TYPE "LBP_typeTMTurret"
TITLE = Tool management / Gestión de herramientas / Werkzeugverwaltung
// User data type for block LBP_TMTurret [DB73] / Tipo de dato de usuario para bloque LBP_TMTurret [DB73] / Anwender-Datentyp für Baustein LBP_TMTurret [DB73]
// stored: IsFailsafeCompliant false
   STRUCT
      IFNo : Array[1..16] of Bool;   // Schnittstelle [Nummer] aktiv / Interface [number] active / Interfaz [número] activa
      Quit : Array[1..16] of Bool;   // Quit-End durchführen / Perform Quit-End / Ejecutar Finalizar confirmación
      TIF : Array[1..16] of Struct
         Comp : Bool;   // Obligatorische Änderung / Compulsory change / Cambio obligatorio
         Perform : Bool;   // Änderung/Wechsel durchführen / Perform change / Ejecutar cambio
         f0_2 : Bool;   // Reserviert / Reserved / Reservado
         T0 : Bool;   // T0 programmiert / T0 programmed / T0 programado
         f0_4 : Bool;   // Reserviert / Reserved / Reservado
         f0_5 : Bool;   // Reserviert / Reserved / Reservado
         ManTOut : Bool;   // Handwerkzeug manuell aus Spindel entladen / Unload hand tool from spindle manually / Descargar a mano herramienta manual del cabezal
         f0_7 : Bool;   // Reserviert / Reserved / Reservado
         PerfStatusError : Bool;   // Negative Quittung / Negative acknowledge / Confirmación negativa
         n1_1 : Bool;   // Reserviert / Reserved / Reservado
         n1_2 : Bool;   // Reserviert / Reserved / Reservado
         n1_3 : Bool;   // Reserviert / Reserved / Reservado
         n1_4 : Bool;   // Reserviert / Reserved / Reservado
         n1_5 : Bool;   // Reserviert / Reserved / Reservado
         n1_6 : Bool;   // Reserviert / Reserved / Reservado
         DataInDB1073 : Bool;   // Multitool-Daten gespeichert in DB1073 / Multitool data stored in DB1073 / Datos Multitool guardados en DB1073
         Channel : Byte;   // Zugeordneter Kanal / Assigned channel / Canal asignado
         TMNo : Byte;   // Werkzeug-Verwaltungsnummer / Tool management number / Número de gestión de herramientas
         VdiTcp0 : DInt;   // Freie Anwendervariable 0 / User parameter 0 / Parámetro de usuario 0
         VdiTcp1 : DInt;   // Freie Anwendervariable 1 / User parameter 1 / Parámetro de usuario 1
         VdiTcp2 : DInt;   // Freie Anwendervariable 2 / User parameter 2 / Parámetro de usuario 2
         BufferIdent : Int;   // Reserviert (Puffer-Identifikation) / Reserved (buffer identification) / Reservado (identificación de búfer)
         BufferNo : Int;   // Rel. Platz im Puffer (res.) / Rel. location in buffer (res.) / Puesto rel. en búfer (res.)
         SMag : Int;   // Magazin-Nummer des Revolvers / Magazine number of turret / Número de almacén del revólver
         SLoc : Int;   // Platznummer für neues Werkzeug / Location number for new tool / Número de puesto para nueva herramienta
         TMag : Int;   // Magazin-Nummer des Revolvers (res.) / Magazine number of turret (res.) / Número de almacén del revólver (res.)
         TLoc : Int;   // Platznummer für vorheriges Werkzeug / Location number for previous tool / Número de puesto para herramienta previa
         LocType : Int;   // Werkzeug neu: Platzart / Tool new: location type / Herramienta nueva: tipo de puesto
         SLeft : Int;   // Werkeug neu: Größe links / Tool new: size left / Herramienta nueva: tamaño izquierda
         SRight : Int;   // Werkeug neu: Größe rechts / Tool new: size right / Herramienta nueva: tamaño derecha
         STop : Int;   // Werkeug neu: Größe oben / Tool new: size top / Herramienta nueva: tamaño arriba
         SBottom : Int;   // Werkeug neu: Größe unten / Tool new: size bottom / Herramienta nueva: tamaño abajo
         TInBuffer : Bool;   // ID für Werkzeuge im Puffer / ID for tools in buffer / ID para herramientas en búfer
         IgnoreDisabled : Bool;   // Deaktiviert ignorieren / Ignore disabled / Ignorar desactivado
         Unload : Bool;   // Zu entladen / To be unloaded / Por descargar
         Load : Bool;   // Zu laden / To be loaded / Por cargar
         MasterTool : Bool;   // Master-Werkzeug / Master tool / Herramienta maestra
         n38_5 : Bool;   // Reserviert / Reserved / Reservado
         Exchange_1to1 : Bool;   // 1:1 Austausch / 1:1 exchange / Cambio 1:1
         HandTool : Bool;   // Handwerkzeug / Hand tool / Herramienta manual
         Active : Bool;   // Aktives Werkzeug / Active tool / Herramienta activa
         Enabled : Bool;   // Werkzeug aktiviert / Tool enabled / Herramienta activada
         Disabled : Bool;   // Werkzeug deaktiviert / Tool disabled / Herramienta desactivada
         Measured : Bool;   // Werkzeug gemessen / Tool measured / Herramienta medida
         Prewarn : Bool;   // Vorwarnungsgrenze erreicht / Prewarning limit reached / Límite de prealarma alcanzado
         Change : Bool;   // Werkzeug wird gewechselt / Tool being changed / Sustituyendo herramienta
         FixedLoc : Bool;   // Werkzeug-Festplatz codiert / Tool fixed location coded / Puesto fijo de herramienta codificado
         Used : Bool;   // Werkzeug war in Gebrauch / Tool was in use / La herramienta estaba en uso
         TNo : Int;   // Werkzeug neu: WZ-Nummer / Tool new: T number / Herramienta nueva: n.º herramienta
         MyPlace : Int;   // Originalplatz des neuen Werkzeugs / Original location of new tool / Puesto de origen de la nueva herramienta
      END_STRUCT;
   END_STRUCT;
   // // TIF[2].Comp : Obligatorische Änderung / Compulsory change / Cambio obligatorio
   // // TIF[3].Comp : Obligatorische Änderung / Compulsory change / Cambio obligatorio
   // // TIF[4].Comp : Obligatorische Änderung / Compulsory change / Cambio obligatorio
   // // TIF[5].Comp : Obligatorische Änderung / Compulsory change / Cambio obligatorio
   // // TIF[6].Comp : Obligatorische Änderung / Compulsory change / Cambio obligatorio
   // // TIF[7].Comp : Obligatorische Änderung / Compulsory change / Cambio obligatorio
   // // TIF[8].Comp : Obligatorische Änderung / Compulsory change / Cambio obligatorio
   // // TIF[9].Comp : Obligatorische Änderung / Compulsory change / Cambio obligatorio
   // // TIF[10].Comp : Obligatorische Änderung / Compulsory change / Cambio obligatorio
   // // TIF[11].Comp : Obligatorische Änderung / Compulsory change / Cambio obligatorio
   // // TIF[12].Comp : Obligatorische Änderung / Compulsory change / Cambio obligatorio
   // // TIF[13].Comp : Obligatorische Änderung / Compulsory change / Cambio obligatorio
   // // TIF[14].Comp : Obligatorische Änderung / Compulsory change / Cambio obligatorio
   // // TIF[15].Comp : Obligatorische Änderung / Compulsory change / Cambio obligatorio
   // // TIF[16].Comp : Obligatorische Änderung / Compulsory change / Cambio obligatorio
   // // TIF[2].Perform : Änderung/Wechsel durchführen / Perform change / Ejecutar cambio
   // // TIF[3].Perform : Änderung/Wechsel durchführen / Perform change / Ejecutar cambio
   // // TIF[4].Perform : Änderung/Wechsel durchführen / Perform change / Ejecutar cambio
   // // TIF[5].Perform : Änderung/Wechsel durchführen / Perform change / Ejecutar cambio
   // // TIF[6].Perform : Änderung/Wechsel durchführen / Perform change / Ejecutar cambio
   // // TIF[7].Perform : Änderung/Wechsel durchführen / Perform change / Ejecutar cambio
   // // TIF[8].Perform : Änderung/Wechsel durchführen / Perform change / Ejecutar cambio
   // // TIF[9].Perform : Änderung/Wechsel durchführen / Perform change / Ejecutar cambio
   // // TIF[10].Perform : Änderung/Wechsel durchführen / Perform change / Ejecutar cambio
   // // TIF[11].Perform : Änderung/Wechsel durchführen / Perform change / Ejecutar cambio
   // // TIF[12].Perform : Änderung/Wechsel durchführen / Perform change / Ejecutar cambio
   // // TIF[13].Perform : Änderung/Wechsel durchführen / Perform change / Ejecutar cambio
   // // TIF[14].Perform : Änderung/Wechsel durchführen / Perform change / Ejecutar cambio
   // // TIF[15].Perform : Änderung/Wechsel durchführen / Perform change / Ejecutar cambio
   // // TIF[16].Perform : Änderung/Wechsel durchführen / Perform change / Ejecutar cambio
   // // TIF[2].f0_2 : Reserviert / Reserved / Reservado
   // // TIF[3].f0_2 : Reserviert / Reserved / Reservado
   // // TIF[4].f0_2 : Reserviert / Reserved / Reservado
   // // TIF[5].f0_2 : Reserviert / Reserved / Reservado
   // // TIF[6].f0_2 : Reserviert / Reserved / Reservado
   // // TIF[7].f0_2 : Reserviert / Reserved / Reservado
   // // TIF[8].f0_2 : Reserviert / Reserved / Reservado
   // // TIF[9].f0_2 : Reserviert / Reserved / Reservado
   // // TIF[10].f0_2 : Reserviert / Reserved / Reservado
   // // TIF[11].f0_2 : Reserviert / Reserved / Reservado
   // // TIF[12].f0_2 : Reserviert / Reserved / Reservado
   // // TIF[13].f0_2 : Reserviert / Reserved / Reservado
   // // TIF[14].f0_2 : Reserviert / Reserved / Reservado
   // // TIF[15].f0_2 : Reserviert / Reserved / Reservado
   // // TIF[16].f0_2 : Reserviert / Reserved / Reservado
   // // TIF[2].T0 : T0 programmiert / T0 programmed / T0 programado
   // // TIF[3].T0 : T0 programmiert / T0 programmed / T0 programado
   // // TIF[4].T0 : T0 programmiert / T0 programmed / T0 programado
   // // TIF[5].T0 : T0 programmiert / T0 programmed / T0 programado
   // // TIF[6].T0 : T0 programmiert / T0 programmed / T0 programado
   // // TIF[7].T0 : T0 programmiert / T0 programmed / T0 programado
   // // TIF[8].T0 : T0 programmiert / T0 programmed / T0 programado
   // // TIF[9].T0 : T0 programmiert / T0 programmed / T0 programado
   // // TIF[10].T0 : T0 programmiert / T0 programmed / T0 programado
   // // TIF[11].T0 : T0 programmiert / T0 programmed / T0 programado
   // // TIF[12].T0 : T0 programmiert / T0 programmed / T0 programado
   // // TIF[13].T0 : T0 programmiert / T0 programmed / T0 programado
   // // TIF[14].T0 : T0 programmiert / T0 programmed / T0 programado
   // // TIF[15].T0 : T0 programmiert / T0 programmed / T0 programado
   // // TIF[16].T0 : T0 programmiert / T0 programmed / T0 programado
   // // TIF[2].f0_4 : Reserviert / Reserved / Reservado
   // // TIF[3].f0_4 : Reserviert / Reserved / Reservado
   // // TIF[4].f0_4 : Reserviert / Reserved / Reservado
   // // TIF[5].f0_4 : Reserviert / Reserved / Reservado
   // // TIF[6].f0_4 : Reserviert / Reserved / Reservado
   // // TIF[7].f0_4 : Reserviert / Reserved / Reservado
   // // TIF[8].f0_4 : Reserviert / Reserved / Reservado
   // // TIF[9].f0_4 : Reserviert / Reserved / Reservado
   // // TIF[10].f0_4 : Reserviert / Reserved / Reservado
   // // TIF[11].f0_4 : Reserviert / Reserved / Reservado
   // // TIF[12].f0_4 : Reserviert / Reserved / Reservado
   // // TIF[13].f0_4 : Reserviert / Reserved / Reservado
   // // TIF[14].f0_4 : Reserviert / Reserved / Reservado
   // // TIF[15].f0_4 : Reserviert / Reserved / Reservado
   // // TIF[16].f0_4 : Reserviert / Reserved / Reservado
   // // TIF[2].f0_5 : Reserviert / Reserved / Reservado
   // // TIF[3].f0_5 : Reserviert / Reserved / Reservado
   // // TIF[4].f0_5 : Reserviert / Reserved / Reservado
   // // TIF[5].f0_5 : Reserviert / Reserved / Reservado
   // // TIF[6].f0_5 : Reserviert / Reserved / Reservado
   // // TIF[7].f0_5 : Reserviert / Reserved / Reservado
   // // TIF[8].f0_5 : Reserviert / Reserved / Reservado
   // // TIF[9].f0_5 : Reserviert / Reserved / Reservado
   // // TIF[10].f0_5 : Reserviert / Reserved / Reservado
   // // TIF[11].f0_5 : Reserviert / Reserved / Reservado
   // // TIF[12].f0_5 : Reserviert / Reserved / Reservado
   // // TIF[13].f0_5 : Reserviert / Reserved / Reservado
   // // TIF[14].f0_5 : Reserviert / Reserved / Reservado
   // // TIF[15].f0_5 : Reserviert / Reserved / Reservado
   // // TIF[16].f0_5 : Reserviert / Reserved / Reservado
   // // TIF[2].ManTOut : Handwerkzeug manuell aus Spindel entladen / Unload hand tool from spindle manually / Descargar a mano herramienta manual del cabezal
   // // TIF[3].ManTOut : Handwerkzeug manuell aus Spindel entladen / Unload hand tool from spindle manually / Descargar a mano herramienta manual del cabezal
   // // TIF[4].ManTOut : Handwerkzeug manuell aus Spindel entladen / Unload hand tool from spindle manually / Descargar a mano herramienta manual del cabezal
   // // TIF[5].ManTOut : Handwerkzeug manuell aus Spindel entladen / Unload hand tool from spindle manually / Descargar a mano herramienta manual del cabezal
   // // TIF[6].ManTOut : Handwerkzeug manuell aus Spindel entladen / Unload hand tool from spindle manually / Descargar a mano herramienta manual del cabezal
   // // TIF[7].ManTOut : Handwerkzeug manuell aus Spindel entladen / Unload hand tool from spindle manually / Descargar a mano herramienta manual del cabezal
   // // TIF[8].ManTOut : Handwerkzeug manuell aus Spindel entladen / Unload hand tool from spindle manually / Descargar a mano herramienta manual del cabezal
   // // TIF[9].ManTOut : Handwerkzeug manuell aus Spindel entladen / Unload hand tool from spindle manually / Descargar a mano herramienta manual del cabezal
   // // TIF[10].ManTOut : Handwerkzeug manuell aus Spindel entladen / Unload hand tool from spindle manually / Descargar a mano herramienta manual del cabezal
   // // TIF[11].ManTOut : Handwerkzeug manuell aus Spindel entladen / Unload hand tool from spindle manually / Descargar a mano herramienta manual del cabezal
   // // TIF[12].ManTOut : Handwerkzeug manuell aus Spindel entladen / Unload hand tool from spindle manually / Descargar a mano herramienta manual del cabezal
   // // TIF[13].ManTOut : Handwerkzeug manuell aus Spindel entladen / Unload hand tool from spindle manually / Descargar a mano herramienta manual del cabezal
   // // TIF[14].ManTOut : Handwerkzeug manuell aus Spindel entladen / Unload hand tool from spindle manually / Descargar a mano herramienta manual del cabezal
   // // TIF[15].ManTOut : Handwerkzeug manuell aus Spindel entladen / Unload hand tool from spindle manually / Descargar a mano herramienta manual del cabezal
   // // TIF[16].ManTOut : Handwerkzeug manuell aus Spindel entladen / Unload hand tool from spindle manually / Descargar a mano herramienta manual del cabezal
   // // TIF[2].f0_7 : Reserviert / Reserved / Reservado
   // // TIF[3].f0_7 : Reserviert / Reserved / Reservado
   // // TIF[4].f0_7 : Reserviert / Reserved / Reservado
   // // TIF[5].f0_7 : Reserviert / Reserved / Reservado
   // // TIF[6].f0_7 : Reserviert / Reserved / Reservado
   // // TIF[7].f0_7 : Reserviert / Reserved / Reservado
   // // TIF[8].f0_7 : Reserviert / Reserved / Reservado
   // // TIF[9].f0_7 : Reserviert / Reserved / Reservado
   // // TIF[10].f0_7 : Reserviert / Reserved / Reservado
   // // TIF[11].f0_7 : Reserviert / Reserved / Reservado
   // // TIF[12].f0_7 : Reserviert / Reserved / Reservado
   // // TIF[13].f0_7 : Reserviert / Reserved / Reservado
   // // TIF[14].f0_7 : Reserviert / Reserved / Reservado
   // // TIF[15].f0_7 : Reserviert / Reserved / Reservado
   // // TIF[16].f0_7 : Reserviert / Reserved / Reservado
   // // TIF[2].PerfStatusError : Negative Quittung / Negative acknowledge / Confirmación negativa
   // // TIF[3].PerfStatusError : Negative Quittung / Negative acknowledge / Confirmación negativa
   // // TIF[4].PerfStatusError : Negative Quittung / Negative acknowledge / Confirmación negativa
   // // TIF[5].PerfStatusError : Negative Quittung / Negative acknowledge / Confirmación negativa
   // // TIF[6].PerfStatusError : Negative Quittung / Negative acknowledge / Confirmación negativa
   // // TIF[7].PerfStatusError : Negative Quittung / Negative acknowledge / Confirmación negativa
   // // TIF[8].PerfStatusError : Negative Quittung / Negative acknowledge / Confirmación negativa
   // // TIF[9].PerfStatusError : Negative Quittung / Negative acknowledge / Confirmación negativa
   // // TIF[10].PerfStatusError : Negative Quittung / Negative acknowledge / Confirmación negativa
   // // TIF[11].PerfStatusError : Negative Quittung / Negative acknowledge / Confirmación negativa
   // // TIF[12].PerfStatusError : Negative Quittung / Negative acknowledge / Confirmación negativa
   // // TIF[13].PerfStatusError : Negative Quittung / Negative acknowledge / Confirmación negativa
   // // TIF[14].PerfStatusError : Negative Quittung / Negative acknowledge / Confirmación negativa
   // // TIF[15].PerfStatusError : Negative Quittung / Negative acknowledge / Confirmación negativa
   // // TIF[16].PerfStatusError : Negative Quittung / Negative acknowledge / Confirmación negativa
   // // TIF[2].n1_1 : Reserviert / Reserved / Reservado
   // // TIF[3].n1_1 : Reserviert / Reserved / Reservado
   // // TIF[4].n1_1 : Reserviert / Reserved / Reservado
   // // TIF[5].n1_1 : Reserviert / Reserved / Reservado
   // // TIF[6].n1_1 : Reserviert / Reserved / Reservado
   // // TIF[7].n1_1 : Reserviert / Reserved / Reservado
   // // TIF[8].n1_1 : Reserviert / Reserved / Reservado
   // // TIF[9].n1_1 : Reserviert / Reserved / Reservado
   // // TIF[10].n1_1 : Reserviert / Reserved / Reservado
   // // TIF[11].n1_1 : Reserviert / Reserved / Reservado
   // // TIF[12].n1_1 : Reserviert / Reserved / Reservado
   // // TIF[13].n1_1 : Reserviert / Reserved / Reservado
   // // TIF[14].n1_1 : Reserviert / Reserved / Reservado
   // // TIF[15].n1_1 : Reserviert / Reserved / Reservado
   // // TIF[16].n1_1 : Reserviert / Reserved / Reservado
   // // TIF[2].n1_2 : Reserviert / Reserved / Reservado
   // // TIF[3].n1_2 : Reserviert / Reserved / Reservado
   // // TIF[4].n1_2 : Reserviert / Reserved / Reservado
   // // TIF[5].n1_2 : Reserviert / Reserved / Reservado
   // // TIF[6].n1_2 : Reserviert / Reserved / Reservado
   // // TIF[7].n1_2 : Reserviert / Reserved / Reservado
   // // TIF[8].n1_2 : Reserviert / Reserved / Reservado
   // // TIF[9].n1_2 : Reserviert / Reserved / Reservado
   // // TIF[10].n1_2 : Reserviert / Reserved / Reservado
   // // TIF[11].n1_2 : Reserviert / Reserved / Reservado
   // // TIF[12].n1_2 : Reserviert / Reserved / Reservado
   // // TIF[13].n1_2 : Reserviert / Reserved / Reservado
   // // TIF[14].n1_2 : Reserviert / Reserved / Reservado
   // // TIF[15].n1_2 : Reserviert / Reserved / Reservado
   // // TIF[16].n1_2 : Reserviert / Reserved / Reservado
   // // TIF[2].n1_3 : Reserviert / Reserved / Reservado
   // // TIF[3].n1_3 : Reserviert / Reserved / Reservado
   // // TIF[4].n1_3 : Reserviert / Reserved / Reservado
   // // TIF[5].n1_3 : Reserviert / Reserved / Reservado
   // // TIF[6].n1_3 : Reserviert / Reserved / Reservado
   // // TIF[7].n1_3 : Reserviert / Reserved / Reservado
   // // TIF[8].n1_3 : Reserviert / Reserved / Reservado
   // // TIF[9].n1_3 : Reserviert / Reserved / Reservado
   // // TIF[10].n1_3 : Reserviert / Reserved / Reservado
   // // TIF[11].n1_3 : Reserviert / Reserved / Reservado
   // // TIF[12].n1_3 : Reserviert / Reserved / Reservado
   // // TIF[13].n1_3 : Reserviert / Reserved / Reservado
   // // TIF[14].n1_3 : Reserviert / Reserved / Reservado
   // // TIF[15].n1_3 : Reserviert / Reserved / Reservado
   // // TIF[16].n1_3 : Reserviert / Reserved / Reservado
   // // TIF[2].n1_4 : Reserviert / Reserved / Reservado
   // // TIF[3].n1_4 : Reserviert / Reserved / Reservado
   // // TIF[4].n1_4 : Reserviert / Reserved / Reservado
   // // TIF[5].n1_4 : Reserviert / Reserved / Reservado
   // // TIF[6].n1_4 : Reserviert / Reserved / Reservado
   // // TIF[7].n1_4 : Reserviert / Reserved / Reservado
   // // TIF[8].n1_4 : Reserviert / Reserved / Reservado
   // // TIF[9].n1_4 : Reserviert / Reserved / Reservado
   // // TIF[10].n1_4 : Reserviert / Reserved / Reservado
   // // TIF[11].n1_4 : Reserviert / Reserved / Reservado
   // // TIF[12].n1_4 : Reserviert / Reserved / Reservado
   // // TIF[13].n1_4 : Reserviert / Reserved / Reservado
   // // TIF[14].n1_4 : Reserviert / Reserved / Reservado
   // // TIF[15].n1_4 : Reserviert / Reserved / Reservado
   // // TIF[16].n1_4 : Reserviert / Reserved / Reservado
   // // TIF[2].n1_5 : Reserviert / Reserved / Reservado
   // // TIF[3].n1_5 : Reserviert / Reserved / Reservado
   // // TIF[4].n1_5 : Reserviert / Reserved / Reservado
   // // TIF[5].n1_5 : Reserviert / Reserved / Reservado
   // // TIF[6].n1_5 : Reserviert / Reserved / Reservado
   // // TIF[7].n1_5 : Reserviert / Reserved / Reservado
   // // TIF[8].n1_5 : Reserviert / Reserved / Reservado
   // // TIF[9].n1_5 : Reserviert / Reserved / Reservado
   // // TIF[10].n1_5 : Reserviert / Reserved / Reservado
   // // TIF[11].n1_5 : Reserviert / Reserved / Reservado
   // // TIF[12].n1_5 : Reserviert / Reserved / Reservado
   // // TIF[13].n1_5 : Reserviert / Reserved / Reservado
   // // TIF[14].n1_5 : Reserviert / Reserved / Reservado
   // // TIF[15].n1_5 : Reserviert / Reserved / Reservado
   // // TIF[16].n1_5 : Reserviert / Reserved / Reservado
   // // TIF[2].n1_6 : Reserviert / Reserved / Reservado
   // // TIF[3].n1_6 : Reserviert / Reserved / Reservado
   // // TIF[4].n1_6 : Reserviert / Reserved / Reservado
   // // TIF[5].n1_6 : Reserviert / Reserved / Reservado
   // // TIF[6].n1_6 : Reserviert / Reserved / Reservado
   // // TIF[7].n1_6 : Reserviert / Reserved / Reservado
   // // TIF[8].n1_6 : Reserviert / Reserved / Reservado
   // // TIF[9].n1_6 : Reserviert / Reserved / Reservado
   // // TIF[10].n1_6 : Reserviert / Reserved / Reservado
   // // TIF[11].n1_6 : Reserviert / Reserved / Reservado
   // // TIF[12].n1_6 : Reserviert / Reserved / Reservado
   // // TIF[13].n1_6 : Reserviert / Reserved / Reservado
   // // TIF[14].n1_6 : Reserviert / Reserved / Reservado
   // // TIF[15].n1_6 : Reserviert / Reserved / Reservado
   // // TIF[16].n1_6 : Reserviert / Reserved / Reservado
   // // TIF[2].DataInDB1073 : Multitool-Daten gespeichert in DB1073 / Multitool data stored in DB1073 / Datos Multitool guardados en DB1073
   // // TIF[3].DataInDB1073 : Multitool-Daten gespeichert in DB1073 / Multitool data stored in DB1073 / Datos Multitool guardados en DB1073
   // // TIF[4].DataInDB1073 : Multitool-Daten gespeichert in DB1073 / Multitool data stored in DB1073 / Datos Multitool guardados en DB1073
   // // TIF[5].DataInDB1073 : Multitool-Daten gespeichert in DB1073 / Multitool data stored in DB1073 / Datos Multitool guardados en DB1073
   // // TIF[6].DataInDB1073 : Multitool-Daten gespeichert in DB1073 / Multitool data stored in DB1073 / Datos Multitool guardados en DB1073
   // // TIF[7].DataInDB1073 : Multitool-Daten gespeichert in DB1073 / Multitool data stored in DB1073 / Datos Multitool guardados en DB1073
   // // TIF[8].DataInDB1073 : Multitool-Daten gespeichert in DB1073 / Multitool data stored in DB1073 / Datos Multitool guardados en DB1073
   // // TIF[9].DataInDB1073 : Multitool-Daten gespeichert in DB1073 / Multitool data stored in DB1073 / Datos Multitool guardados en DB1073
   // // TIF[10].DataInDB1073 : Multitool-Daten gespeichert in DB1073 / Multitool data stored in DB1073 / Datos Multitool guardados en DB1073
   // // TIF[11].DataInDB1073 : Multitool-Daten gespeichert in DB1073 / Multitool data stored in DB1073 / Datos Multitool guardados en DB1073
   // // TIF[12].DataInDB1073 : Multitool-Daten gespeichert in DB1073 / Multitool data stored in DB1073 / Datos Multitool guardados en DB1073
   // // TIF[13].DataInDB1073 : Multitool-Daten gespeichert in DB1073 / Multitool data stored in DB1073 / Datos Multitool guardados en DB1073
   // // TIF[14].DataInDB1073 : Multitool-Daten gespeichert in DB1073 / Multitool data stored in DB1073 / Datos Multitool guardados en DB1073
   // // TIF[15].DataInDB1073 : Multitool-Daten gespeichert in DB1073 / Multitool data stored in DB1073 / Datos Multitool guardados en DB1073
   // // TIF[16].DataInDB1073 : Multitool-Daten gespeichert in DB1073 / Multitool data stored in DB1073 / Datos Multitool guardados en DB1073
   // // TIF[2].Channel : Zugeordneter Kanal / Assigned channel / Canal asignado
   // // TIF[3].Channel : Zugeordneter Kanal / Assigned channel / Canal asignado
   // // TIF[4].Channel : Zugeordneter Kanal / Assigned channel / Canal asignado
   // // TIF[5].Channel : Zugeordneter Kanal / Assigned channel / Canal asignado
   // // TIF[6].Channel : Zugeordneter Kanal / Assigned channel / Canal asignado
   // // TIF[7].Channel : Zugeordneter Kanal / Assigned channel / Canal asignado
   // // TIF[8].Channel : Zugeordneter Kanal / Assigned channel / Canal asignado
   // // TIF[9].Channel : Zugeordneter Kanal / Assigned channel / Canal asignado
   // // TIF[10].Channel : Zugeordneter Kanal / Assigned channel / Canal asignado
   // // TIF[11].Channel : Zugeordneter Kanal / Assigned channel / Canal asignado
   // // TIF[12].Channel : Zugeordneter Kanal / Assigned channel / Canal asignado
   // // TIF[13].Channel : Zugeordneter Kanal / Assigned channel / Canal asignado
   // // TIF[14].Channel : Zugeordneter Kanal / Assigned channel / Canal asignado
   // // TIF[15].Channel : Zugeordneter Kanal / Assigned channel / Canal asignado
   // // TIF[16].Channel : Zugeordneter Kanal / Assigned channel / Canal asignado
   // // TIF[2].TMNo : Werkzeug-Verwaltungsnummer / Tool management number / Número de gestión de herramientas
   // // TIF[3].TMNo : Werkzeug-Verwaltungsnummer / Tool management number / Número de gestión de herramientas
   // // TIF[4].TMNo : Werkzeug-Verwaltungsnummer / Tool management number / Número de gestión de herramientas
   // // TIF[5].TMNo : Werkzeug-Verwaltungsnummer / Tool management number / Número de gestión de herramientas
   // // TIF[6].TMNo : Werkzeug-Verwaltungsnummer / Tool management number / Número de gestión de herramientas
   // // TIF[7].TMNo : Werkzeug-Verwaltungsnummer / Tool management number / Número de gestión de herramientas
   // // TIF[8].TMNo : Werkzeug-Verwaltungsnummer / Tool management number / Número de gestión de herramientas
   // // TIF[9].TMNo : Werkzeug-Verwaltungsnummer / Tool management number / Número de gestión de herramientas
   // // TIF[10].TMNo : Werkzeug-Verwaltungsnummer / Tool management number / Número de gestión de herramientas
   // // TIF[11].TMNo : Werkzeug-Verwaltungsnummer / Tool management number / Número de gestión de herramientas
   // // TIF[12].TMNo : Werkzeug-Verwaltungsnummer / Tool management number / Número de gestión de herramientas
   // // TIF[13].TMNo : Werkzeug-Verwaltungsnummer / Tool management number / Número de gestión de herramientas
   // // TIF[14].TMNo : Werkzeug-Verwaltungsnummer / Tool management number / Número de gestión de herramientas
   // // TIF[15].TMNo : Werkzeug-Verwaltungsnummer / Tool management number / Número de gestión de herramientas
   // // TIF[16].TMNo : Werkzeug-Verwaltungsnummer / Tool management number / Número de gestión de herramientas
   // // TIF[2].VdiTcp0 : Freie Anwendervariable 0 / User parameter 0 / Parámetro de usuario 0
   // // TIF[3].VdiTcp0 : Freie Anwendervariable 0 / User parameter 0 / Parámetro de usuario 0
   // // TIF[4].VdiTcp0 : Freie Anwendervariable 0 / User parameter 0 / Parámetro de usuario 0
   // // TIF[5].VdiTcp0 : Freie Anwendervariable 0 / User parameter 0 / Parámetro de usuario 0
   // // TIF[6].VdiTcp0 : Freie Anwendervariable 0 / User parameter 0 / Parámetro de usuario 0
   // // TIF[7].VdiTcp0 : Freie Anwendervariable 0 / User parameter 0 / Parámetro de usuario 0
   // // TIF[8].VdiTcp0 : Freie Anwendervariable 0 / User parameter 0 / Parámetro de usuario 0
   // // TIF[9].VdiTcp0 : Freie Anwendervariable 0 / User parameter 0 / Parámetro de usuario 0
   // // TIF[10].VdiTcp0 : Freie Anwendervariable 0 / User parameter 0 / Parámetro de usuario 0
   // // TIF[11].VdiTcp0 : Freie Anwendervariable 0 / User parameter 0 / Parámetro de usuario 0
   // // TIF[12].VdiTcp0 : Freie Anwendervariable 0 / User parameter 0 / Parámetro de usuario 0
   // // TIF[13].VdiTcp0 : Freie Anwendervariable 0 / User parameter 0 / Parámetro de usuario 0
   // // TIF[14].VdiTcp0 : Freie Anwendervariable 0 / User parameter 0 / Parámetro de usuario 0
   // // TIF[15].VdiTcp0 : Freie Anwendervariable 0 / User parameter 0 / Parámetro de usuario 0
   // // TIF[16].VdiTcp0 : Freie Anwendervariable 0 / User parameter 0 / Parámetro de usuario 0
   // // TIF[2].VdiTcp1 : Freie Anwendervariable 1 / User parameter 1 / Parámetro de usuario 1
   // // TIF[3].VdiTcp1 : Freie Anwendervariable 1 / User parameter 1 / Parámetro de usuario 1
   // // TIF[4].VdiTcp1 : Freie Anwendervariable 1 / User parameter 1 / Parámetro de usuario 1
   // // TIF[5].VdiTcp1 : Freie Anwendervariable 1 / User parameter 1 / Parámetro de usuario 1
   // // TIF[6].VdiTcp1 : Freie Anwendervariable 1 / User parameter 1 / Parámetro de usuario 1
   // // TIF[7].VdiTcp1 : Freie Anwendervariable 1 / User parameter 1 / Parámetro de usuario 1
   // // TIF[8].VdiTcp1 : Freie Anwendervariable 1 / User parameter 1 / Parámetro de usuario 1
   // // TIF[9].VdiTcp1 : Freie Anwendervariable 1 / User parameter 1 / Parámetro de usuario 1
   // // TIF[10].VdiTcp1 : Freie Anwendervariable 1 / User parameter 1 / Parámetro de usuario 1
   // // TIF[11].VdiTcp1 : Freie Anwendervariable 1 / User parameter 1 / Parámetro de usuario 1
   // // TIF[12].VdiTcp1 : Freie Anwendervariable 1 / User parameter 1 / Parámetro de usuario 1
   // // TIF[13].VdiTcp1 : Freie Anwendervariable 1 / User parameter 1 / Parámetro de usuario 1
   // // TIF[14].VdiTcp1 : Freie Anwendervariable 1 / User parameter 1 / Parámetro de usuario 1
   // // TIF[15].VdiTcp1 : Freie Anwendervariable 1 / User parameter 1 / Parámetro de usuario 1
   // // TIF[16].VdiTcp1 : Freie Anwendervariable 1 / User parameter 1 / Parámetro de usuario 1
   // // TIF[2].VdiTcp2 : Freie Anwendervariable 2 / User parameter 2 / Parámetro de usuario 2
   // // TIF[3].VdiTcp2 : Freie Anwendervariable 2 / User parameter 2 / Parámetro de usuario 2
   // // TIF[4].VdiTcp2 : Freie Anwendervariable 2 / User parameter 2 / Parámetro de usuario 2
   // // TIF[5].VdiTcp2 : Freie Anwendervariable 2 / User parameter 2 / Parámetro de usuario 2
   // // TIF[6].VdiTcp2 : Freie Anwendervariable 2 / User parameter 2 / Parámetro de usuario 2
   // // TIF[7].VdiTcp2 : Freie Anwendervariable 2 / User parameter 2 / Parámetro de usuario 2
   // // TIF[8].VdiTcp2 : Freie Anwendervariable 2 / User parameter 2 / Parámetro de usuario 2
   // // TIF[9].VdiTcp2 : Freie Anwendervariable 2 / User parameter 2 / Parámetro de usuario 2
   // // TIF[10].VdiTcp2 : Freie Anwendervariable 2 / User parameter 2 / Parámetro de usuario 2
   // // TIF[11].VdiTcp2 : Freie Anwendervariable 2 / User parameter 2 / Parámetro de usuario 2
   // // TIF[12].VdiTcp2 : Freie Anwendervariable 2 / User parameter 2 / Parámetro de usuario 2
   // // TIF[13].VdiTcp2 : Freie Anwendervariable 2 / User parameter 2 / Parámetro de usuario 2
   // // TIF[14].VdiTcp2 : Freie Anwendervariable 2 / User parameter 2 / Parámetro de usuario 2
   // // TIF[15].VdiTcp2 : Freie Anwendervariable 2 / User parameter 2 / Parámetro de usuario 2
   // // TIF[16].VdiTcp2 : Freie Anwendervariable 2 / User parameter 2 / Parámetro de usuario 2
   // // TIF[2].BufferIdent : Reserviert (Puffer-Identifikation) / Reserved (buffer identification) / Reservado (identificación de búfer)
   // // TIF[3].BufferIdent : Reserviert (Puffer-Identifikation) / Reserved (buffer identification) / Reservado (identificación de búfer)
   // // TIF[4].BufferIdent : Reserviert (Puffer-Identifikation) / Reserved (buffer identification) / Reservado (identificación de búfer)
   // // TIF[5].BufferIdent : Reserviert (Puffer-Identifikation) / Reserved (buffer identification) / Reservado (identificación de búfer)
   // // TIF[6].BufferIdent : Reserviert (Puffer-Identifikation) / Reserved (buffer identification) / Reservado (identificación de búfer)
   // // TIF[7].BufferIdent : Reserviert (Puffer-Identifikation) / Reserved (buffer identification) / Reservado (identificación de búfer)
   // // TIF[8].BufferIdent : Reserviert (Puffer-Identifikation) / Reserved (buffer identification) / Reservado (identificación de búfer)
   // // TIF[9].BufferIdent : Reserviert (Puffer-Identifikation) / Reserved (buffer identification) / Reservado (identificación de búfer)
   // // TIF[10].BufferIdent : Reserviert (Puffer-Identifikation) / Reserved (buffer identification) / Reservado (identificación de búfer)
   // // TIF[11].BufferIdent : Reserviert (Puffer-Identifikation) / Reserved (buffer identification) / Reservado (identificación de búfer)
   // // TIF[12].BufferIdent : Reserviert (Puffer-Identifikation) / Reserved (buffer identification) / Reservado (identificación de búfer)
   // // TIF[13].BufferIdent : Reserviert (Puffer-Identifikation) / Reserved (buffer identification) / Reservado (identificación de búfer)
   // // TIF[14].BufferIdent : Reserviert (Puffer-Identifikation) / Reserved (buffer identification) / Reservado (identificación de búfer)
   // // TIF[15].BufferIdent : Reserviert (Puffer-Identifikation) / Reserved (buffer identification) / Reservado (identificación de búfer)
   // // TIF[16].BufferIdent : Reserviert (Puffer-Identifikation) / Reserved (buffer identification) / Reservado (identificación de búfer)
   // // TIF[2].BufferNo : Rel. Platz im Puffer (res.) / Rel. location in buffer (res.) / Puesto rel. en búfer (res.)
   // // TIF[3].BufferNo : Rel. Platz im Puffer (res.) / Rel. location in buffer (res.) / Puesto rel. en búfer (res.)
   // // TIF[4].BufferNo : Rel. Platz im Puffer (res.) / Rel. location in buffer (res.) / Puesto rel. en búfer (res.)
   // // TIF[5].BufferNo : Rel. Platz im Puffer (res.) / Rel. location in buffer (res.) / Puesto rel. en búfer (res.)
   // // TIF[6].BufferNo : Rel. Platz im Puffer (res.) / Rel. location in buffer (res.) / Puesto rel. en búfer (res.)
   // // TIF[7].BufferNo : Rel. Platz im Puffer (res.) / Rel. location in buffer (res.) / Puesto rel. en búfer (res.)
   // // TIF[8].BufferNo : Rel. Platz im Puffer (res.) / Rel. location in buffer (res.) / Puesto rel. en búfer (res.)
   // // TIF[9].BufferNo : Rel. Platz im Puffer (res.) / Rel. location in buffer (res.) / Puesto rel. en búfer (res.)
   // // TIF[10].BufferNo : Rel. Platz im Puffer (res.) / Rel. location in buffer (res.) / Puesto rel. en búfer (res.)
   // // TIF[11].BufferNo : Rel. Platz im Puffer (res.) / Rel. location in buffer (res.) / Puesto rel. en búfer (res.)
   // // TIF[12].BufferNo : Rel. Platz im Puffer (res.) / Rel. location in buffer (res.) / Puesto rel. en búfer (res.)
   // // TIF[13].BufferNo : Rel. Platz im Puffer (res.) / Rel. location in buffer (res.) / Puesto rel. en búfer (res.)
   // // TIF[14].BufferNo : Rel. Platz im Puffer (res.) / Rel. location in buffer (res.) / Puesto rel. en búfer (res.)
   // // TIF[15].BufferNo : Rel. Platz im Puffer (res.) / Rel. location in buffer (res.) / Puesto rel. en búfer (res.)
   // // TIF[16].BufferNo : Rel. Platz im Puffer (res.) / Rel. location in buffer (res.) / Puesto rel. en búfer (res.)
   // // TIF[2].SMag : Magazin-Nummer des Revolvers / Magazine number of turret / Número de almacén del revólver
   // // TIF[3].SMag : Magazin-Nummer des Revolvers / Magazine number of turret / Número de almacén del revólver
   // // TIF[4].SMag : Magazin-Nummer des Revolvers / Magazine number of turret / Número de almacén del revólver
   // // TIF[5].SMag : Magazin-Nummer des Revolvers / Magazine number of turret / Número de almacén del revólver
   // // TIF[6].SMag : Magazin-Nummer des Revolvers / Magazine number of turret / Número de almacén del revólver
   // // TIF[7].SMag : Magazin-Nummer des Revolvers / Magazine number of turret / Número de almacén del revólver
   // // TIF[8].SMag : Magazin-Nummer des Revolvers / Magazine number of turret / Número de almacén del revólver
   // // TIF[9].SMag : Magazin-Nummer des Revolvers / Magazine number of turret / Número de almacén del revólver
   // // TIF[10].SMag : Magazin-Nummer des Revolvers / Magazine number of turret / Número de almacén del revólver
   // // TIF[11].SMag : Magazin-Nummer des Revolvers / Magazine number of turret / Número de almacén del revólver
   // // TIF[12].SMag : Magazin-Nummer des Revolvers / Magazine number of turret / Número de almacén del revólver
   // // TIF[13].SMag : Magazin-Nummer des Revolvers / Magazine number of turret / Número de almacén del revólver
   // // TIF[14].SMag : Magazin-Nummer des Revolvers / Magazine number of turret / Número de almacén del revólver
   // // TIF[15].SMag : Magazin-Nummer des Revolvers / Magazine number of turret / Número de almacén del revólver
   // // TIF[16].SMag : Magazin-Nummer des Revolvers / Magazine number of turret / Número de almacén del revólver
   // // TIF[2].SLoc : Platznummer für neues Werkzeug / Location number for new tool / Número de puesto para nueva herramienta
   // // TIF[3].SLoc : Platznummer für neues Werkzeug / Location number for new tool / Número de puesto para nueva herramienta
   // // TIF[4].SLoc : Platznummer für neues Werkzeug / Location number for new tool / Número de puesto para nueva herramienta
   // // TIF[5].SLoc : Platznummer für neues Werkzeug / Location number for new tool / Número de puesto para nueva herramienta
   // // TIF[6].SLoc : Platznummer für neues Werkzeug / Location number for new tool / Número de puesto para nueva herramienta
   // // TIF[7].SLoc : Platznummer für neues Werkzeug / Location number for new tool / Número de puesto para nueva herramienta
   // // TIF[8].SLoc : Platznummer für neues Werkzeug / Location number for new tool / Número de puesto para nueva herramienta
   // // TIF[9].SLoc : Platznummer für neues Werkzeug / Location number for new tool / Número de puesto para nueva herramienta
   // // TIF[10].SLoc : Platznummer für neues Werkzeug / Location number for new tool / Número de puesto para nueva herramienta
   // // TIF[11].SLoc : Platznummer für neues Werkzeug / Location number for new tool / Número de puesto para nueva herramienta
   // // TIF[12].SLoc : Platznummer für neues Werkzeug / Location number for new tool / Número de puesto para nueva herramienta
   // // TIF[13].SLoc : Platznummer für neues Werkzeug / Location number for new tool / Número de puesto para nueva herramienta
   // // TIF[14].SLoc : Platznummer für neues Werkzeug / Location number for new tool / Número de puesto para nueva herramienta
   // // TIF[15].SLoc : Platznummer für neues Werkzeug / Location number for new tool / Número de puesto para nueva herramienta
   // // TIF[16].SLoc : Platznummer für neues Werkzeug / Location number for new tool / Número de puesto para nueva herramienta
   // // TIF[2].TMag : Magazin-Nummer des Revolvers (res.) / Magazine number of turret (res.) / Número de almacén del revólver (res.)
   // // TIF[3].TMag : Magazin-Nummer des Revolvers (res.) / Magazine number of turret (res.) / Número de almacén del revólver (res.)
   // // TIF[4].TMag : Magazin-Nummer des Revolvers (res.) / Magazine number of turret (res.) / Número de almacén del revólver (res.)
   // // TIF[5].TMag : Magazin-Nummer des Revolvers (res.) / Magazine number of turret (res.) / Número de almacén del revólver (res.)
   // // TIF[6].TMag : Magazin-Nummer des Revolvers (res.) / Magazine number of turret (res.) / Número de almacén del revólver (res.)
   // // TIF[7].TMag : Magazin-Nummer des Revolvers (res.) / Magazine number of turret (res.) / Número de almacén del revólver (res.)
   // // TIF[8].TMag : Magazin-Nummer des Revolvers (res.) / Magazine number of turret (res.) / Número de almacén del revólver (res.)
   // // TIF[9].TMag : Magazin-Nummer des Revolvers (res.) / Magazine number of turret (res.) / Número de almacén del revólver (res.)
   // // TIF[10].TMag : Magazin-Nummer des Revolvers (res.) / Magazine number of turret (res.) / Número de almacén del revólver (res.)
   // // TIF[11].TMag : Magazin-Nummer des Revolvers (res.) / Magazine number of turret (res.) / Número de almacén del revólver (res.)
   // // TIF[12].TMag : Magazin-Nummer des Revolvers (res.) / Magazine number of turret (res.) / Número de almacén del revólver (res.)
   // // TIF[13].TMag : Magazin-Nummer des Revolvers (res.) / Magazine number of turret (res.) / Número de almacén del revólver (res.)
   // // TIF[14].TMag : Magazin-Nummer des Revolvers (res.) / Magazine number of turret (res.) / Número de almacén del revólver (res.)
   // // TIF[15].TMag : Magazin-Nummer des Revolvers (res.) / Magazine number of turret (res.) / Número de almacén del revólver (res.)
   // // TIF[16].TMag : Magazin-Nummer des Revolvers (res.) / Magazine number of turret (res.) / Número de almacén del revólver (res.)
   // // TIF[2].TLoc : Platznummer für vorheriges Werkzeug / Location number for previous tool / Número de puesto para herramienta previa
   // // TIF[3].TLoc : Platznummer für vorheriges Werkzeug / Location number for previous tool / Número de puesto para herramienta previa
   // // TIF[4].TLoc : Platznummer für vorheriges Werkzeug / Location number for previous tool / Número de puesto para herramienta previa
   // // TIF[5].TLoc : Platznummer für vorheriges Werkzeug / Location number for previous tool / Número de puesto para herramienta previa
   // // TIF[6].TLoc : Platznummer für vorheriges Werkzeug / Location number for previous tool / Número de puesto para herramienta previa
   // // TIF[7].TLoc : Platznummer für vorheriges Werkzeug / Location number for previous tool / Número de puesto para herramienta previa
   // // TIF[8].TLoc : Platznummer für vorheriges Werkzeug / Location number for previous tool / Número de puesto para herramienta previa
   // // TIF[9].TLoc : Platznummer für vorheriges Werkzeug / Location number for previous tool / Número de puesto para herramienta previa
   // // TIF[10].TLoc : Platznummer für vorheriges Werkzeug / Location number for previous tool / Número de puesto para herramienta previa
   // // TIF[11].TLoc : Platznummer für vorheriges Werkzeug / Location number for previous tool / Número de puesto para herramienta previa
   // // TIF[12].TLoc : Platznummer für vorheriges Werkzeug / Location number for previous tool / Número de puesto para herramienta previa
   // // TIF[13].TLoc : Platznummer für vorheriges Werkzeug / Location number for previous tool / Número de puesto para herramienta previa
   // // TIF[14].TLoc : Platznummer für vorheriges Werkzeug / Location number for previous tool / Número de puesto para herramienta previa
   // // TIF[15].TLoc : Platznummer für vorheriges Werkzeug / Location number for previous tool / Número de puesto para herramienta previa
   // // TIF[16].TLoc : Platznummer für vorheriges Werkzeug / Location number for previous tool / Número de puesto para herramienta previa
   // // TIF[2].LocType : Werkzeug neu: Platzart / Tool new: location type / Herramienta nueva: tipo de puesto
   // // TIF[3].LocType : Werkzeug neu: Platzart / Tool new: location type / Herramienta nueva: tipo de puesto
   // // TIF[4].LocType : Werkzeug neu: Platzart / Tool new: location type / Herramienta nueva: tipo de puesto
   // // TIF[5].LocType : Werkzeug neu: Platzart / Tool new: location type / Herramienta nueva: tipo de puesto
   // // TIF[6].LocType : Werkzeug neu: Platzart / Tool new: location type / Herramienta nueva: tipo de puesto
   // // TIF[7].LocType : Werkzeug neu: Platzart / Tool new: location type / Herramienta nueva: tipo de puesto
   // // TIF[8].LocType : Werkzeug neu: Platzart / Tool new: location type / Herramienta nueva: tipo de puesto
   // // TIF[9].LocType : Werkzeug neu: Platzart / Tool new: location type / Herramienta nueva: tipo de puesto
   // // TIF[10].LocType : Werkzeug neu: Platzart / Tool new: location type / Herramienta nueva: tipo de puesto
   // // TIF[11].LocType : Werkzeug neu: Platzart / Tool new: location type / Herramienta nueva: tipo de puesto
   // // TIF[12].LocType : Werkzeug neu: Platzart / Tool new: location type / Herramienta nueva: tipo de puesto
   // // TIF[13].LocType : Werkzeug neu: Platzart / Tool new: location type / Herramienta nueva: tipo de puesto
   // // TIF[14].LocType : Werkzeug neu: Platzart / Tool new: location type / Herramienta nueva: tipo de puesto
   // // TIF[15].LocType : Werkzeug neu: Platzart / Tool new: location type / Herramienta nueva: tipo de puesto
   // // TIF[16].LocType : Werkzeug neu: Platzart / Tool new: location type / Herramienta nueva: tipo de puesto
   // // TIF[2].SLeft : Werkeug neu: Größe links / Tool new: size left / Herramienta nueva: tamaño izquierda
   // // TIF[3].SLeft : Werkeug neu: Größe links / Tool new: size left / Herramienta nueva: tamaño izquierda
   // // TIF[4].SLeft : Werkeug neu: Größe links / Tool new: size left / Herramienta nueva: tamaño izquierda
   // // TIF[5].SLeft : Werkeug neu: Größe links / Tool new: size left / Herramienta nueva: tamaño izquierda
   // // TIF[6].SLeft : Werkeug neu: Größe links / Tool new: size left / Herramienta nueva: tamaño izquierda
   // // TIF[7].SLeft : Werkeug neu: Größe links / Tool new: size left / Herramienta nueva: tamaño izquierda
   // // TIF[8].SLeft : Werkeug neu: Größe links / Tool new: size left / Herramienta nueva: tamaño izquierda
   // // TIF[9].SLeft : Werkeug neu: Größe links / Tool new: size left / Herramienta nueva: tamaño izquierda
   // // TIF[10].SLeft : Werkeug neu: Größe links / Tool new: size left / Herramienta nueva: tamaño izquierda
   // // TIF[11].SLeft : Werkeug neu: Größe links / Tool new: size left / Herramienta nueva: tamaño izquierda
   // // TIF[12].SLeft : Werkeug neu: Größe links / Tool new: size left / Herramienta nueva: tamaño izquierda
   // // TIF[13].SLeft : Werkeug neu: Größe links / Tool new: size left / Herramienta nueva: tamaño izquierda
   // // TIF[14].SLeft : Werkeug neu: Größe links / Tool new: size left / Herramienta nueva: tamaño izquierda
   // // TIF[15].SLeft : Werkeug neu: Größe links / Tool new: size left / Herramienta nueva: tamaño izquierda
   // // TIF[16].SLeft : Werkeug neu: Größe links / Tool new: size left / Herramienta nueva: tamaño izquierda
   // // TIF[2].SRight : Werkeug neu: Größe rechts / Tool new: size right / Herramienta nueva: tamaño derecha
   // // TIF[3].SRight : Werkeug neu: Größe rechts / Tool new: size right / Herramienta nueva: tamaño derecha
   // // TIF[4].SRight : Werkeug neu: Größe rechts / Tool new: size right / Herramienta nueva: tamaño derecha
   // // TIF[5].SRight : Werkeug neu: Größe rechts / Tool new: size right / Herramienta nueva: tamaño derecha
   // // TIF[6].SRight : Werkeug neu: Größe rechts / Tool new: size right / Herramienta nueva: tamaño derecha
   // // TIF[7].SRight : Werkeug neu: Größe rechts / Tool new: size right / Herramienta nueva: tamaño derecha
   // // TIF[8].SRight : Werkeug neu: Größe rechts / Tool new: size right / Herramienta nueva: tamaño derecha
   // // TIF[9].SRight : Werkeug neu: Größe rechts / Tool new: size right / Herramienta nueva: tamaño derecha
   // // TIF[10].SRight : Werkeug neu: Größe rechts / Tool new: size right / Herramienta nueva: tamaño derecha
   // // TIF[11].SRight : Werkeug neu: Größe rechts / Tool new: size right / Herramienta nueva: tamaño derecha
   // // TIF[12].SRight : Werkeug neu: Größe rechts / Tool new: size right / Herramienta nueva: tamaño derecha
   // // TIF[13].SRight : Werkeug neu: Größe rechts / Tool new: size right / Herramienta nueva: tamaño derecha
   // // TIF[14].SRight : Werkeug neu: Größe rechts / Tool new: size right / Herramienta nueva: tamaño derecha
   // // TIF[15].SRight : Werkeug neu: Größe rechts / Tool new: size right / Herramienta nueva: tamaño derecha
   // // TIF[16].SRight : Werkeug neu: Größe rechts / Tool new: size right / Herramienta nueva: tamaño derecha
   // // TIF[2].STop : Werkeug neu: Größe oben / Tool new: size top / Herramienta nueva: tamaño arriba
   // // TIF[3].STop : Werkeug neu: Größe oben / Tool new: size top / Herramienta nueva: tamaño arriba
   // // TIF[4].STop : Werkeug neu: Größe oben / Tool new: size top / Herramienta nueva: tamaño arriba
   // // TIF[5].STop : Werkeug neu: Größe oben / Tool new: size top / Herramienta nueva: tamaño arriba
   // // TIF[6].STop : Werkeug neu: Größe oben / Tool new: size top / Herramienta nueva: tamaño arriba
   // // TIF[7].STop : Werkeug neu: Größe oben / Tool new: size top / Herramienta nueva: tamaño arriba
   // // TIF[8].STop : Werkeug neu: Größe oben / Tool new: size top / Herramienta nueva: tamaño arriba
   // // TIF[9].STop : Werkeug neu: Größe oben / Tool new: size top / Herramienta nueva: tamaño arriba
   // // TIF[10].STop : Werkeug neu: Größe oben / Tool new: size top / Herramienta nueva: tamaño arriba
   // // TIF[11].STop : Werkeug neu: Größe oben / Tool new: size top / Herramienta nueva: tamaño arriba
   // // TIF[12].STop : Werkeug neu: Größe oben / Tool new: size top / Herramienta nueva: tamaño arriba
   // // TIF[13].STop : Werkeug neu: Größe oben / Tool new: size top / Herramienta nueva: tamaño arriba
   // // TIF[14].STop : Werkeug neu: Größe oben / Tool new: size top / Herramienta nueva: tamaño arriba
   // // TIF[15].STop : Werkeug neu: Größe oben / Tool new: size top / Herramienta nueva: tamaño arriba
   // // TIF[16].STop : Werkeug neu: Größe oben / Tool new: size top / Herramienta nueva: tamaño arriba
   // // TIF[2].SBottom : Werkeug neu: Größe unten / Tool new: size bottom / Herramienta nueva: tamaño abajo
   // // TIF[3].SBottom : Werkeug neu: Größe unten / Tool new: size bottom / Herramienta nueva: tamaño abajo
   // // TIF[4].SBottom : Werkeug neu: Größe unten / Tool new: size bottom / Herramienta nueva: tamaño abajo
   // // TIF[5].SBottom : Werkeug neu: Größe unten / Tool new: size bottom / Herramienta nueva: tamaño abajo
   // // TIF[6].SBottom : Werkeug neu: Größe unten / Tool new: size bottom / Herramienta nueva: tamaño abajo
   // // TIF[7].SBottom : Werkeug neu: Größe unten / Tool new: size bottom / Herramienta nueva: tamaño abajo
   // // TIF[8].SBottom : Werkeug neu: Größe unten / Tool new: size bottom / Herramienta nueva: tamaño abajo
   // // TIF[9].SBottom : Werkeug neu: Größe unten / Tool new: size bottom / Herramienta nueva: tamaño abajo
   // // TIF[10].SBottom : Werkeug neu: Größe unten / Tool new: size bottom / Herramienta nueva: tamaño abajo
   // // TIF[11].SBottom : Werkeug neu: Größe unten / Tool new: size bottom / Herramienta nueva: tamaño abajo
   // // TIF[12].SBottom : Werkeug neu: Größe unten / Tool new: size bottom / Herramienta nueva: tamaño abajo
   // // TIF[13].SBottom : Werkeug neu: Größe unten / Tool new: size bottom / Herramienta nueva: tamaño abajo
   // // TIF[14].SBottom : Werkeug neu: Größe unten / Tool new: size bottom / Herramienta nueva: tamaño abajo
   // // TIF[15].SBottom : Werkeug neu: Größe unten / Tool new: size bottom / Herramienta nueva: tamaño abajo
   // // TIF[16].SBottom : Werkeug neu: Größe unten / Tool new: size bottom / Herramienta nueva: tamaño abajo
   // // TIF[2].TInBuffer : ID für Werkzeuge im Puffer / ID for tools in buffer / ID para herramientas en búfer
   // // TIF[3].TInBuffer : ID für Werkzeuge im Puffer / ID for tools in buffer / ID para herramientas en búfer
   // // TIF[4].TInBuffer : ID für Werkzeuge im Puffer / ID for tools in buffer / ID para herramientas en búfer
   // // TIF[5].TInBuffer : ID für Werkzeuge im Puffer / ID for tools in buffer / ID para herramientas en búfer
   // // TIF[6].TInBuffer : ID für Werkzeuge im Puffer / ID for tools in buffer / ID para herramientas en búfer
   // // TIF[7].TInBuffer : ID für Werkzeuge im Puffer / ID for tools in buffer / ID para herramientas en búfer
   // // TIF[8].TInBuffer : ID für Werkzeuge im Puffer / ID for tools in buffer / ID para herramientas en búfer
   // // TIF[9].TInBuffer : ID für Werkzeuge im Puffer / ID for tools in buffer / ID para herramientas en búfer
   // // TIF[10].TInBuffer : ID für Werkzeuge im Puffer / ID for tools in buffer / ID para herramientas en búfer
   // // TIF[11].TInBuffer : ID für Werkzeuge im Puffer / ID for tools in buffer / ID para herramientas en búfer
   // // TIF[12].TInBuffer : ID für Werkzeuge im Puffer / ID for tools in buffer / ID para herramientas en búfer
   // // TIF[13].TInBuffer : ID für Werkzeuge im Puffer / ID for tools in buffer / ID para herramientas en búfer
   // // TIF[14].TInBuffer : ID für Werkzeuge im Puffer / ID for tools in buffer / ID para herramientas en búfer
   // // TIF[15].TInBuffer : ID für Werkzeuge im Puffer / ID for tools in buffer / ID para herramientas en búfer
   // // TIF[16].TInBuffer : ID für Werkzeuge im Puffer / ID for tools in buffer / ID para herramientas en búfer
   // // TIF[2].IgnoreDisabled : Deaktiviert ignorieren / Ignore disabled / Ignorar desactivado
   // // TIF[3].IgnoreDisabled : Deaktiviert ignorieren / Ignore disabled / Ignorar desactivado
   // // TIF[4].IgnoreDisabled : Deaktiviert ignorieren / Ignore disabled / Ignorar desactivado
   // // TIF[5].IgnoreDisabled : Deaktiviert ignorieren / Ignore disabled / Ignorar desactivado
   // // TIF[6].IgnoreDisabled : Deaktiviert ignorieren / Ignore disabled / Ignorar desactivado
   // // TIF[7].IgnoreDisabled : Deaktiviert ignorieren / Ignore disabled / Ignorar desactivado
   // // TIF[8].IgnoreDisabled : Deaktiviert ignorieren / Ignore disabled / Ignorar desactivado
   // // TIF[9].IgnoreDisabled : Deaktiviert ignorieren / Ignore disabled / Ignorar desactivado
   // // TIF[10].IgnoreDisabled : Deaktiviert ignorieren / Ignore disabled / Ignorar desactivado
   // // TIF[11].IgnoreDisabled : Deaktiviert ignorieren / Ignore disabled / Ignorar desactivado
   // // TIF[12].IgnoreDisabled : Deaktiviert ignorieren / Ignore disabled / Ignorar desactivado
   // // TIF[13].IgnoreDisabled : Deaktiviert ignorieren / Ignore disabled / Ignorar desactivado
   // // TIF[14].IgnoreDisabled : Deaktiviert ignorieren / Ignore disabled / Ignorar desactivado
   // // TIF[15].IgnoreDisabled : Deaktiviert ignorieren / Ignore disabled / Ignorar desactivado
   // // TIF[16].IgnoreDisabled : Deaktiviert ignorieren / Ignore disabled / Ignorar desactivado
   // // TIF[2].Unload : Zu entladen / To be unloaded / Por descargar
   // // TIF[3].Unload : Zu entladen / To be unloaded / Por descargar
   // // TIF[4].Unload : Zu entladen / To be unloaded / Por descargar
   // // TIF[5].Unload : Zu entladen / To be unloaded / Por descargar
   // // TIF[6].Unload : Zu entladen / To be unloaded / Por descargar
   // // TIF[7].Unload : Zu entladen / To be unloaded / Por descargar
   // // TIF[8].Unload : Zu entladen / To be unloaded / Por descargar
   // // TIF[9].Unload : Zu entladen / To be unloaded / Por descargar
   // // TIF[10].Unload : Zu entladen / To be unloaded / Por descargar
   // // TIF[11].Unload : Zu entladen / To be unloaded / Por descargar
   // // TIF[12].Unload : Zu entladen / To be unloaded / Por descargar
   // // TIF[13].Unload : Zu entladen / To be unloaded / Por descargar
   // // TIF[14].Unload : Zu entladen / To be unloaded / Por descargar
   // // TIF[15].Unload : Zu entladen / To be unloaded / Por descargar
   // // TIF[16].Unload : Zu entladen / To be unloaded / Por descargar
   // // TIF[2].Load : Zu laden / To be loaded / Por cargar
   // // TIF[3].Load : Zu laden / To be loaded / Por cargar
   // // TIF[4].Load : Zu laden / To be loaded / Por cargar
   // // TIF[5].Load : Zu laden / To be loaded / Por cargar
   // // TIF[6].Load : Zu laden / To be loaded / Por cargar
   // // TIF[7].Load : Zu laden / To be loaded / Por cargar
   // // TIF[8].Load : Zu laden / To be loaded / Por cargar
   // // TIF[9].Load : Zu laden / To be loaded / Por cargar
   // // TIF[10].Load : Zu laden / To be loaded / Por cargar
   // // TIF[11].Load : Zu laden / To be loaded / Por cargar
   // // TIF[12].Load : Zu laden / To be loaded / Por cargar
   // // TIF[13].Load : Zu laden / To be loaded / Por cargar
   // // TIF[14].Load : Zu laden / To be loaded / Por cargar
   // // TIF[15].Load : Zu laden / To be loaded / Por cargar
   // // TIF[16].Load : Zu laden / To be loaded / Por cargar
   // // TIF[2].MasterTool : Master-Werkzeug / Master tool / Herramienta maestra
   // // TIF[3].MasterTool : Master-Werkzeug / Master tool / Herramienta maestra
   // // TIF[4].MasterTool : Master-Werkzeug / Master tool / Herramienta maestra
   // // TIF[5].MasterTool : Master-Werkzeug / Master tool / Herramienta maestra
   // // TIF[6].MasterTool : Master-Werkzeug / Master tool / Herramienta maestra
   // // TIF[7].MasterTool : Master-Werkzeug / Master tool / Herramienta maestra
   // // TIF[8].MasterTool : Master-Werkzeug / Master tool / Herramienta maestra
   // // TIF[9].MasterTool : Master-Werkzeug / Master tool / Herramienta maestra
   // // TIF[10].MasterTool : Master-Werkzeug / Master tool / Herramienta maestra
   // // TIF[11].MasterTool : Master-Werkzeug / Master tool / Herramienta maestra
   // // TIF[12].MasterTool : Master-Werkzeug / Master tool / Herramienta maestra
   // // TIF[13].MasterTool : Master-Werkzeug / Master tool / Herramienta maestra
   // // TIF[14].MasterTool : Master-Werkzeug / Master tool / Herramienta maestra
   // // TIF[15].MasterTool : Master-Werkzeug / Master tool / Herramienta maestra
   // // TIF[16].MasterTool : Master-Werkzeug / Master tool / Herramienta maestra
   // // TIF[2].n38_5 : Reserviert / Reserved / Reservado
   // // TIF[3].n38_5 : Reserviert / Reserved / Reservado
   // // TIF[4].n38_5 : Reserviert / Reserved / Reservado
   // // TIF[5].n38_5 : Reserviert / Reserved / Reservado
   // // TIF[6].n38_5 : Reserviert / Reserved / Reservado
   // // TIF[7].n38_5 : Reserviert / Reserved / Reservado
   // // TIF[8].n38_5 : Reserviert / Reserved / Reservado
   // // TIF[9].n38_5 : Reserviert / Reserved / Reservado
   // // TIF[10].n38_5 : Reserviert / Reserved / Reservado
   // // TIF[11].n38_5 : Reserviert / Reserved / Reservado
   // // TIF[12].n38_5 : Reserviert / Reserved / Reservado
   // // TIF[13].n38_5 : Reserviert / Reserved / Reservado
   // // TIF[14].n38_5 : Reserviert / Reserved / Reservado
   // // TIF[15].n38_5 : Reserviert / Reserved / Reservado
   // // TIF[16].n38_5 : Reserviert / Reserved / Reservado
   // // TIF[2].Exchange_1to1 : 1:1 Austausch / 1:1 exchange / Cambio 1:1
   // // TIF[3].Exchange_1to1 : 1:1 Austausch / 1:1 exchange / Cambio 1:1
   // // TIF[4].Exchange_1to1 : 1:1 Austausch / 1:1 exchange / Cambio 1:1
   // // TIF[5].Exchange_1to1 : 1:1 Austausch / 1:1 exchange / Cambio 1:1
   // // TIF[6].Exchange_1to1 : 1:1 Austausch / 1:1 exchange / Cambio 1:1
   // // TIF[7].Exchange_1to1 : 1:1 Austausch / 1:1 exchange / Cambio 1:1
   // // TIF[8].Exchange_1to1 : 1:1 Austausch / 1:1 exchange / Cambio 1:1
   // // TIF[9].Exchange_1to1 : 1:1 Austausch / 1:1 exchange / Cambio 1:1
   // // TIF[10].Exchange_1to1 : 1:1 Austausch / 1:1 exchange / Cambio 1:1
   // // TIF[11].Exchange_1to1 : 1:1 Austausch / 1:1 exchange / Cambio 1:1
   // // TIF[12].Exchange_1to1 : 1:1 Austausch / 1:1 exchange / Cambio 1:1
   // // TIF[13].Exchange_1to1 : 1:1 Austausch / 1:1 exchange / Cambio 1:1
   // // TIF[14].Exchange_1to1 : 1:1 Austausch / 1:1 exchange / Cambio 1:1
   // // TIF[15].Exchange_1to1 : 1:1 Austausch / 1:1 exchange / Cambio 1:1
   // // TIF[16].Exchange_1to1 : 1:1 Austausch / 1:1 exchange / Cambio 1:1
   // // TIF[2].HandTool : Handwerkzeug / Hand tool / Herramienta manual
   // // TIF[3].HandTool : Handwerkzeug / Hand tool / Herramienta manual
   // // TIF[4].HandTool : Handwerkzeug / Hand tool / Herramienta manual
   // // TIF[5].HandTool : Handwerkzeug / Hand tool / Herramienta manual
   // // TIF[6].HandTool : Handwerkzeug / Hand tool / Herramienta manual
   // // TIF[7].HandTool : Handwerkzeug / Hand tool / Herramienta manual
   // // TIF[8].HandTool : Handwerkzeug / Hand tool / Herramienta manual
   // // TIF[9].HandTool : Handwerkzeug / Hand tool / Herramienta manual
   // // TIF[10].HandTool : Handwerkzeug / Hand tool / Herramienta manual
   // // TIF[11].HandTool : Handwerkzeug / Hand tool / Herramienta manual
   // // TIF[12].HandTool : Handwerkzeug / Hand tool / Herramienta manual
   // // TIF[13].HandTool : Handwerkzeug / Hand tool / Herramienta manual
   // // TIF[14].HandTool : Handwerkzeug / Hand tool / Herramienta manual
   // // TIF[15].HandTool : Handwerkzeug / Hand tool / Herramienta manual
   // // TIF[16].HandTool : Handwerkzeug / Hand tool / Herramienta manual
   // // TIF[2].Active : Aktives Werkzeug / Active tool / Herramienta activa
   // // TIF[3].Active : Aktives Werkzeug / Active tool / Herramienta activa
   // // TIF[4].Active : Aktives Werkzeug / Active tool / Herramienta activa
   // // TIF[5].Active : Aktives Werkzeug / Active tool / Herramienta activa
   // // TIF[6].Active : Aktives Werkzeug / Active tool / Herramienta activa
   // // TIF[7].Active : Aktives Werkzeug / Active tool / Herramienta activa
   // // TIF[8].Active : Aktives Werkzeug / Active tool / Herramienta activa
   // // TIF[9].Active : Aktives Werkzeug / Active tool / Herramienta activa
   // // TIF[10].Active : Aktives Werkzeug / Active tool / Herramienta activa
   // // TIF[11].Active : Aktives Werkzeug / Active tool / Herramienta activa
   // // TIF[12].Active : Aktives Werkzeug / Active tool / Herramienta activa
   // // TIF[13].Active : Aktives Werkzeug / Active tool / Herramienta activa
   // // TIF[14].Active : Aktives Werkzeug / Active tool / Herramienta activa
   // // TIF[15].Active : Aktives Werkzeug / Active tool / Herramienta activa
   // // TIF[16].Active : Aktives Werkzeug / Active tool / Herramienta activa
   // // TIF[2].Enabled : Werkzeug aktiviert / Tool enabled / Herramienta activada
   // // TIF[3].Enabled : Werkzeug aktiviert / Tool enabled / Herramienta activada
   // // TIF[4].Enabled : Werkzeug aktiviert / Tool enabled / Herramienta activada
   // // TIF[5].Enabled : Werkzeug aktiviert / Tool enabled / Herramienta activada
   // // TIF[6].Enabled : Werkzeug aktiviert / Tool enabled / Herramienta activada
   // // TIF[7].Enabled : Werkzeug aktiviert / Tool enabled / Herramienta activada
   // // TIF[8].Enabled : Werkzeug aktiviert / Tool enabled / Herramienta activada
   // // TIF[9].Enabled : Werkzeug aktiviert / Tool enabled / Herramienta activada
   // // TIF[10].Enabled : Werkzeug aktiviert / Tool enabled / Herramienta activada
   // // TIF[11].Enabled : Werkzeug aktiviert / Tool enabled / Herramienta activada
   // // TIF[12].Enabled : Werkzeug aktiviert / Tool enabled / Herramienta activada
   // // TIF[13].Enabled : Werkzeug aktiviert / Tool enabled / Herramienta activada
   // // TIF[14].Enabled : Werkzeug aktiviert / Tool enabled / Herramienta activada
   // // TIF[15].Enabled : Werkzeug aktiviert / Tool enabled / Herramienta activada
   // // TIF[16].Enabled : Werkzeug aktiviert / Tool enabled / Herramienta activada
   // // TIF[2].Disabled : Werkzeug deaktiviert / Tool disabled / Herramienta desactivada
   // // TIF[3].Disabled : Werkzeug deaktiviert / Tool disabled / Herramienta desactivada
   // // TIF[4].Disabled : Werkzeug deaktiviert / Tool disabled / Herramienta desactivada
   // // TIF[5].Disabled : Werkzeug deaktiviert / Tool disabled / Herramienta desactivada
   // // TIF[6].Disabled : Werkzeug deaktiviert / Tool disabled / Herramienta desactivada
   // // TIF[7].Disabled : Werkzeug deaktiviert / Tool disabled / Herramienta desactivada
   // // TIF[8].Disabled : Werkzeug deaktiviert / Tool disabled / Herramienta desactivada
   // // TIF[9].Disabled : Werkzeug deaktiviert / Tool disabled / Herramienta desactivada
   // // TIF[10].Disabled : Werkzeug deaktiviert / Tool disabled / Herramienta desactivada
   // // TIF[11].Disabled : Werkzeug deaktiviert / Tool disabled / Herramienta desactivada
   // // TIF[12].Disabled : Werkzeug deaktiviert / Tool disabled / Herramienta desactivada
   // // TIF[13].Disabled : Werkzeug deaktiviert / Tool disabled / Herramienta desactivada
   // // TIF[14].Disabled : Werkzeug deaktiviert / Tool disabled / Herramienta desactivada
   // // TIF[15].Disabled : Werkzeug deaktiviert / Tool disabled / Herramienta desactivada
   // // TIF[16].Disabled : Werkzeug deaktiviert / Tool disabled / Herramienta desactivada
   // // TIF[2].Measured : Werkzeug gemessen / Tool measured / Herramienta medida
   // // TIF[3].Measured : Werkzeug gemessen / Tool measured / Herramienta medida
   // // TIF[4].Measured : Werkzeug gemessen / Tool measured / Herramienta medida
   // // TIF[5].Measured : Werkzeug gemessen / Tool measured / Herramienta medida
   // // TIF[6].Measured : Werkzeug gemessen / Tool measured / Herramienta medida
   // // TIF[7].Measured : Werkzeug gemessen / Tool measured / Herramienta medida
   // // TIF[8].Measured : Werkzeug gemessen / Tool measured / Herramienta medida
   // // TIF[9].Measured : Werkzeug gemessen / Tool measured / Herramienta medida
   // // TIF[10].Measured : Werkzeug gemessen / Tool measured / Herramienta medida
   // // TIF[11].Measured : Werkzeug gemessen / Tool measured / Herramienta medida
   // // TIF[12].Measured : Werkzeug gemessen / Tool measured / Herramienta medida
   // // TIF[13].Measured : Werkzeug gemessen / Tool measured / Herramienta medida
   // // TIF[14].Measured : Werkzeug gemessen / Tool measured / Herramienta medida
   // // TIF[15].Measured : Werkzeug gemessen / Tool measured / Herramienta medida
   // // TIF[16].Measured : Werkzeug gemessen / Tool measured / Herramienta medida
   // // TIF[2].Prewarn : Vorwarnungsgrenze erreicht / Prewarning limit reached / Límite de prealarma alcanzado
   // // TIF[3].Prewarn : Vorwarnungsgrenze erreicht / Prewarning limit reached / Límite de prealarma alcanzado
   // // TIF[4].Prewarn : Vorwarnungsgrenze erreicht / Prewarning limit reached / Límite de prealarma alcanzado
   // // TIF[5].Prewarn : Vorwarnungsgrenze erreicht / Prewarning limit reached / Límite de prealarma alcanzado
   // // TIF[6].Prewarn : Vorwarnungsgrenze erreicht / Prewarning limit reached / Límite de prealarma alcanzado
   // // TIF[7].Prewarn : Vorwarnungsgrenze erreicht / Prewarning limit reached / Límite de prealarma alcanzado
   // // TIF[8].Prewarn : Vorwarnungsgrenze erreicht / Prewarning limit reached / Límite de prealarma alcanzado
   // // TIF[9].Prewarn : Vorwarnungsgrenze erreicht / Prewarning limit reached / Límite de prealarma alcanzado
   // // TIF[10].Prewarn : Vorwarnungsgrenze erreicht / Prewarning limit reached / Límite de prealarma alcanzado
   // // TIF[11].Prewarn : Vorwarnungsgrenze erreicht / Prewarning limit reached / Límite de prealarma alcanzado
   // // TIF[12].Prewarn : Vorwarnungsgrenze erreicht / Prewarning limit reached / Límite de prealarma alcanzado
   // // TIF[13].Prewarn : Vorwarnungsgrenze erreicht / Prewarning limit reached / Límite de prealarma alcanzado
   // // TIF[14].Prewarn : Vorwarnungsgrenze erreicht / Prewarning limit reached / Límite de prealarma alcanzado
   // // TIF[15].Prewarn : Vorwarnungsgrenze erreicht / Prewarning limit reached / Límite de prealarma alcanzado
   // // TIF[16].Prewarn : Vorwarnungsgrenze erreicht / Prewarning limit reached / Límite de prealarma alcanzado
   // // TIF[2].Change : Werkzeug wird gewechselt / Tool being changed / Sustituyendo herramienta
   // // TIF[3].Change : Werkzeug wird gewechselt / Tool being changed / Sustituyendo herramienta
   // // TIF[4].Change : Werkzeug wird gewechselt / Tool being changed / Sustituyendo herramienta
   // // TIF[5].Change : Werkzeug wird gewechselt / Tool being changed / Sustituyendo herramienta
   // // TIF[6].Change : Werkzeug wird gewechselt / Tool being changed / Sustituyendo herramienta
   // // TIF[7].Change : Werkzeug wird gewechselt / Tool being changed / Sustituyendo herramienta
   // // TIF[8].Change : Werkzeug wird gewechselt / Tool being changed / Sustituyendo herramienta
   // // TIF[9].Change : Werkzeug wird gewechselt / Tool being changed / Sustituyendo herramienta
   // // TIF[10].Change : Werkzeug wird gewechselt / Tool being changed / Sustituyendo herramienta
   // // TIF[11].Change : Werkzeug wird gewechselt / Tool being changed / Sustituyendo herramienta
   // // TIF[12].Change : Werkzeug wird gewechselt / Tool being changed / Sustituyendo herramienta
   // // TIF[13].Change : Werkzeug wird gewechselt / Tool being changed / Sustituyendo herramienta
   // // TIF[14].Change : Werkzeug wird gewechselt / Tool being changed / Sustituyendo herramienta
   // // TIF[15].Change : Werkzeug wird gewechselt / Tool being changed / Sustituyendo herramienta
   // // TIF[16].Change : Werkzeug wird gewechselt / Tool being changed / Sustituyendo herramienta
   // // TIF[2].FixedLoc : Werkzeug-Festplatz codiert / Tool fixed location coded / Puesto fijo de herramienta codificado
   // // TIF[3].FixedLoc : Werkzeug-Festplatz codiert / Tool fixed location coded / Puesto fijo de herramienta codificado
   // // TIF[4].FixedLoc : Werkzeug-Festplatz codiert / Tool fixed location coded / Puesto fijo de herramienta codificado
   // // TIF[5].FixedLoc : Werkzeug-Festplatz codiert / Tool fixed location coded / Puesto fijo de herramienta codificado
   // // TIF[6].FixedLoc : Werkzeug-Festplatz codiert / Tool fixed location coded / Puesto fijo de herramienta codificado
   // // TIF[7].FixedLoc : Werkzeug-Festplatz codiert / Tool fixed location coded / Puesto fijo de herramienta codificado
   // // TIF[8].FixedLoc : Werkzeug-Festplatz codiert / Tool fixed location coded / Puesto fijo de herramienta codificado
   // // TIF[9].FixedLoc : Werkzeug-Festplatz codiert / Tool fixed location coded / Puesto fijo de herramienta codificado
   // // TIF[10].FixedLoc : Werkzeug-Festplatz codiert / Tool fixed location coded / Puesto fijo de herramienta codificado
   // // TIF[11].FixedLoc : Werkzeug-Festplatz codiert / Tool fixed location coded / Puesto fijo de herramienta codificado
   // // TIF[12].FixedLoc : Werkzeug-Festplatz codiert / Tool fixed location coded / Puesto fijo de herramienta codificado
   // // TIF[13].FixedLoc : Werkzeug-Festplatz codiert / Tool fixed location coded / Puesto fijo de herramienta codificado
   // // TIF[14].FixedLoc : Werkzeug-Festplatz codiert / Tool fixed location coded / Puesto fijo de herramienta codificado
   // // TIF[15].FixedLoc : Werkzeug-Festplatz codiert / Tool fixed location coded / Puesto fijo de herramienta codificado
   // // TIF[16].FixedLoc : Werkzeug-Festplatz codiert / Tool fixed location coded / Puesto fijo de herramienta codificado
   // // TIF[2].Used : Werkzeug war in Gebrauch / Tool was in use / La herramienta estaba en uso
   // // TIF[3].Used : Werkzeug war in Gebrauch / Tool was in use / La herramienta estaba en uso
   // // TIF[4].Used : Werkzeug war in Gebrauch / Tool was in use / La herramienta estaba en uso
   // // TIF[5].Used : Werkzeug war in Gebrauch / Tool was in use / La herramienta estaba en uso
   // // TIF[6].Used : Werkzeug war in Gebrauch / Tool was in use / La herramienta estaba en uso
   // // TIF[7].Used : Werkzeug war in Gebrauch / Tool was in use / La herramienta estaba en uso
   // // TIF[8].Used : Werkzeug war in Gebrauch / Tool was in use / La herramienta estaba en uso
   // // TIF[9].Used : Werkzeug war in Gebrauch / Tool was in use / La herramienta estaba en uso
   // // TIF[10].Used : Werkzeug war in Gebrauch / Tool was in use / La herramienta estaba en uso
   // // TIF[11].Used : Werkzeug war in Gebrauch / Tool was in use / La herramienta estaba en uso
   // // TIF[12].Used : Werkzeug war in Gebrauch / Tool was in use / La herramienta estaba en uso
   // // TIF[13].Used : Werkzeug war in Gebrauch / Tool was in use / La herramienta estaba en uso
   // // TIF[14].Used : Werkzeug war in Gebrauch / Tool was in use / La herramienta estaba en uso
   // // TIF[15].Used : Werkzeug war in Gebrauch / Tool was in use / La herramienta estaba en uso
   // // TIF[16].Used : Werkzeug war in Gebrauch / Tool was in use / La herramienta estaba en uso
   // // TIF[2].TNo : Werkzeug neu: WZ-Nummer / Tool new: T number / Herramienta nueva: n.º herramienta
   // // TIF[3].TNo : Werkzeug neu: WZ-Nummer / Tool new: T number / Herramienta nueva: n.º herramienta
   // // TIF[4].TNo : Werkzeug neu: WZ-Nummer / Tool new: T number / Herramienta nueva: n.º herramienta
   // // TIF[5].TNo : Werkzeug neu: WZ-Nummer / Tool new: T number / Herramienta nueva: n.º herramienta
   // // TIF[6].TNo : Werkzeug neu: WZ-Nummer / Tool new: T number / Herramienta nueva: n.º herramienta
   // // TIF[7].TNo : Werkzeug neu: WZ-Nummer / Tool new: T number / Herramienta nueva: n.º herramienta
   // // TIF[8].TNo : Werkzeug neu: WZ-Nummer / Tool new: T number / Herramienta nueva: n.º herramienta
   // // TIF[9].TNo : Werkzeug neu: WZ-Nummer / Tool new: T number / Herramienta nueva: n.º herramienta
   // // TIF[10].TNo : Werkzeug neu: WZ-Nummer / Tool new: T number / Herramienta nueva: n.º herramienta
   // // TIF[11].TNo : Werkzeug neu: WZ-Nummer / Tool new: T number / Herramienta nueva: n.º herramienta
   // // TIF[12].TNo : Werkzeug neu: WZ-Nummer / Tool new: T number / Herramienta nueva: n.º herramienta
   // // TIF[13].TNo : Werkzeug neu: WZ-Nummer / Tool new: T number / Herramienta nueva: n.º herramienta
   // // TIF[14].TNo : Werkzeug neu: WZ-Nummer / Tool new: T number / Herramienta nueva: n.º herramienta
   // // TIF[15].TNo : Werkzeug neu: WZ-Nummer / Tool new: T number / Herramienta nueva: n.º herramienta
   // // TIF[16].TNo : Werkzeug neu: WZ-Nummer / Tool new: T number / Herramienta nueva: n.º herramienta
   // // TIF[2].MyPlace : Originalplatz des neuen Werkzeugs / Original location of new tool / Puesto de origen de la nueva herramienta
   // // TIF[3].MyPlace : Originalplatz des neuen Werkzeugs / Original location of new tool / Puesto de origen de la nueva herramienta
   // // TIF[4].MyPlace : Originalplatz des neuen Werkzeugs / Original location of new tool / Puesto de origen de la nueva herramienta
   // // TIF[5].MyPlace : Originalplatz des neuen Werkzeugs / Original location of new tool / Puesto de origen de la nueva herramienta
   // // TIF[6].MyPlace : Originalplatz des neuen Werkzeugs / Original location of new tool / Puesto de origen de la nueva herramienta
   // // TIF[7].MyPlace : Originalplatz des neuen Werkzeugs / Original location of new tool / Puesto de origen de la nueva herramienta
   // // TIF[8].MyPlace : Originalplatz des neuen Werkzeugs / Original location of new tool / Puesto de origen de la nueva herramienta
   // // TIF[9].MyPlace : Originalplatz des neuen Werkzeugs / Original location of new tool / Puesto de origen de la nueva herramienta
   // // TIF[10].MyPlace : Originalplatz des neuen Werkzeugs / Original location of new tool / Puesto de origen de la nueva herramienta
   // // TIF[11].MyPlace : Originalplatz des neuen Werkzeugs / Original location of new tool / Puesto de origen de la nueva herramienta
   // // TIF[12].MyPlace : Originalplatz des neuen Werkzeugs / Original location of new tool / Puesto de origen de la nueva herramienta
   // // TIF[13].MyPlace : Originalplatz des neuen Werkzeugs / Original location of new tool / Puesto de origen de la nueva herramienta
   // // TIF[14].MyPlace : Originalplatz des neuen Werkzeugs / Original location of new tool / Puesto de origen de la nueva herramienta
   // // TIF[15].MyPlace : Originalplatz des neuen Werkzeugs / Original location of new tool / Puesto de origen de la nueva herramienta
   // // TIF[16].MyPlace : Originalplatz des neuen Werkzeugs / Original location of new tool / Puesto de origen de la nueva herramienta
END_TYPE

